INTERFACE IInspector EXTENDS TcoCore.ITcoTaskStatus

PROPERTY Result : eInspectorResult
GET
END_GET
END_PROPERTY

END_INTERFACE

(* stored: Version 1.1.0.1, ProductVersion 3.1.4024.9
   Itf IInspector: Id {0cbe9e39-d5a4-05af-17ce-7965efd20de3}
   Property Result: Id {059b95a9-368b-016b-1e77-bc829a9a2a15}
   Get Get: Id {11bcb09e-df05-0600-3fcc-c1e8eab49bfc} *)
